// SIMATIC S7-200 project (STEP 7-Micro/WIN), CPU 224 CN REL 02.01

ORGANIZATION_BLOCK 主程序:OB1
TITLE=程序注释
BEGIN
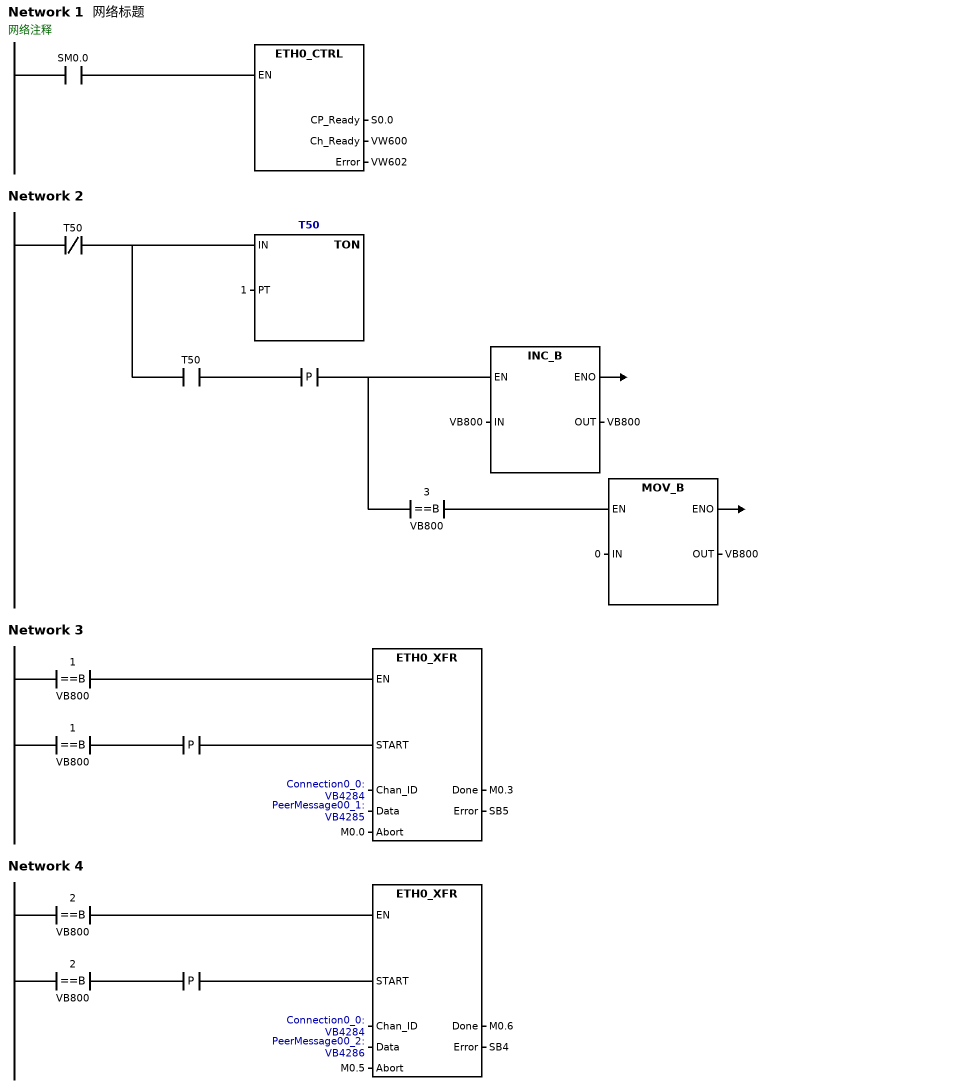
Network 1 // 网络标题
// 网络注释
LD     SM0.0
CALL   ETH0_CTRL:SBR1, S0.0, VW600, VW602
Network 2
LDN    T50
TON    T50, 1
A      T50
EU
INCB   VB800
AB=    3, VB800
MOVB   0, VB800
Network 3
LDB=   1, VB800
=      L60.0
LDB=   1, VB800
EU
=      L63.7
LD     L60.0
CALL   ETH0_XFR:SBR2, L63.7, Connection0_0:VB4284, PeerMessage00_1:VB4285, M0.0, M0.3, SB5
Network 4
LDB=   2, VB800
=      L60.0
LDB=   2, VB800
EU
=      L63.7
LD     L60.0
CALL   ETH0_XFR:SBR2, L63.7, Connection0_0:VB4284, PeerMessage00_2:VB4286, M0.5, M0.6, SB4
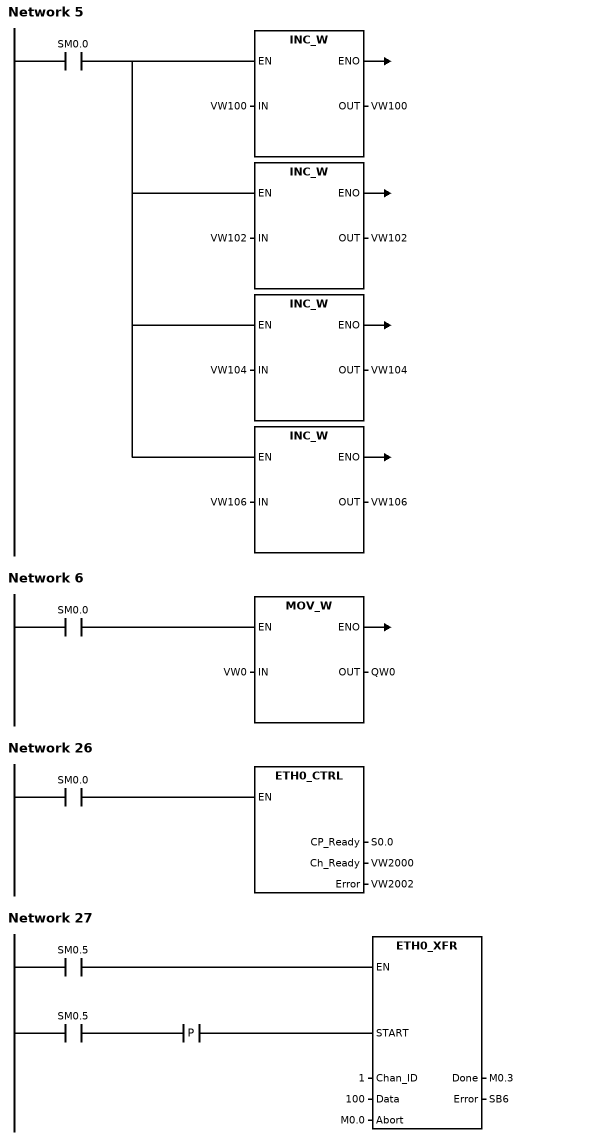
Network 5
LD     SM0.0
INCW   VW100
INCW   VW102
INCW   VW104
INCW   VW106
Network 6
LD     SM0.0
MOVW   VW0, QW0
Network 26
LD     SM0.0
CALL   ETH0_CTRL:SBR1, S0.0, VW2000, VW2002
Network 27
LD     SM0.5
=      L60.0
LD     SM0.5
EU
=      L63.7
LD     L60.0
CALL   ETH0_XFR:SBR2, L63.7, 1, 100, M0.0, M0.3, SB6
END_ORGANIZATION_BLOCK

// SBR1: protected block, not included

// SBR2: protected block, not included

// (further data pages could not be read)
